VISUALIZATION FrameDummy  // 2x2
END_VISUALIZATION

(* stored: Version 1.1.0.1, ProductVersion 3.1.4024.9
   Visu FrameDummy: Id {feb9971a-9636-405d-89be-7fd78b31aef0} *)
